{attribute 'qualified_only'}
VAR_GLOBAL PERSISTENT
	EventBuffer 					: ARRAY [1..500] OF ST_Event;
	Part_is_Sorted					: BOOL;
END_VAR

(* stored: Version 1.1.0.1, ProductVersion 3.1.4024.12
   GVL GVL: Id {8a814bb3-96b5-4f0e-a827-550052e1e8f4} *)
